PROGRAM MAIN
VAR
	PL1_FU1_BGB1 AT %I* : BOOL;
END_VAR

END_PROGRAM

(* stored: Version 1.1.0.1, ProductVersion 3.1.4024.11
   POU MAIN: Id {4bae149f-6428-4d71-830f-ae86950d85bf}, SpecialFunc None *)
